// TIA Portal project "SCL_V13_SP1_1" (V13)

(* hardware
DEVICE "ET 200S-Station_1"  ET 200S station
   slot 0: "Baugruppenträger_0"  Rail
   slot 2: "PLC_1"  IM151-8 CPU  6ES7 151-8AB00-0AB0  V2.7
      slot 1: "PROFINET-Schnittstelle_1"  PN-IO
         slot 1: "Port_1"  Port
         slot 2: "Port_2"  Port
         slot 3: "Port_3"  Port
   slot 4: "PM-E DC24V_1"  PM-E 24VDC  6ES7 138-4CA01-0AA0
   slot 5: "4AI x I 2WIRE ST_1"  4AI x I 2WIRE ST  6ES7 134-4GD00-0AB0
   slot 6: "2AO x U ST_1"  2AO x U ST  6ES7 135-4FB01-0AB0
   slot 7: "8DI x DC24V_1"  8DI x 24VDC  6ES7 131-4BF00-0AA0
   slot 8: "8DI x DC24V_2"  8DI x 24VDC  6ES7 131-4BF00-0AA0
   slot 9: "8DI x DC24V_3"  8DI x 24VDC  6ES7 131-4BF00-0AA0
   slot 10: "8DI x DC24V_4"  8DI x 24VDC  6ES7 131-4BF00-0AA0
   slot 11: "8DO x DC24V / 0,5A_1"  8DO x 24VDC / 0.5A  6ES7 132-4BF00-0AA0
   slot 12: "8DO x DC24V / 0,5A_2"  8DO x 24VDC / 0.5A  6ES7 132-4BF00-0AA0
   slot 13: "8DO x DC24V / 0,5A_3"  8DO x 24VDC / 0.5A  6ES7 132-4BF00-0AA0
   slot 14: "8DO x DC24V / 0,5A_4"  8DO x 24VDC / 0.5A  6ES7 132-4BF00-0AA0
DEVICE "HMI_1"  TP 177B 6" PN/DP
   slot 0: "HMI"  HMI  6AV6 642-0BA01-1AX1  11.0.2.0
   slot 1: "HMI_RT_1"  TP 177B 6" PN/DP  6AV6 642-0BA01-1AX1  11.0.2.0
   slot 5: "HMI_1.IE_CP_1"  PROFINET Schnittstelle
      slot 1: "PROFINET Schnittstelle_1"  PROFINET Schnittstelle
         slot 1: "Port_1"  Port
   slot 7: "HMI_1.MPI/DP_CP_1"  MPI/DP Schnittstelle
DEVICE "PC-System_1"  SIMATIC PC station
   slot 0: "SIMATIC PC-Station"  Rail  SIMATIC PC-Station  V1.0
      slot 125: "Stationmanager"  Station_Manager  V6.0.4
   slot 1: "IE Allgemein_1"  IE General  IE_CP  V8.2.0
   slot 2: "HMI_RT_2"  WinCC RT Advanced  6AV2 104-0xxxx-xxxx  13.0.0.0
*)

// ===== PLC "PLC_1"  IM151-8 CPU =====

VAR_GLOBAL   // PLC tag table "Standard-Variablentabelle"
   "Volumen_Kugel" AT %MD10 : Real;
   "Tag_1" AT %MD20 : Real;
   "Sensor" AT %EW272 : Int;
   "Zu_gross" AT %M3.0 : Bool;
   "Abstand" AT %MD60 : Real;
   "Bit" AT %M0.0 : Bool;
   "Status_scale" AT %MW64 : Word;
   "Test" AT %MD66 : Real;
   "Zaehleingang" AT %E3.0 : Bool;
   "Ueber_PV" AT %M0.1 : Bool;
   "Zaehlerausgang" AT %MW26 : Int;
END_VAR

DATA_BLOCK "Datenbaustein_1"   // DB1
{ S7_Optimized_Access := 'FALSE' }
VERSION : 0.1
   VAR
      Datenspeicher : Array[1..2, 1..10] of Real;
   END_VAR
BEGIN
END_DATA_BLOCK

DATA_BLOCK "Daten_lesen_schreiben_DB"   // DB2
{ S7_Optimized_Access := 'FALSE' }
VERSION : 0.1
// stored: InstanceOfName Daten_lesen_schreiben
"Daten_lesen_schreiben"
BEGIN
END_DATA_BLOCK

FUNCTION_BLOCK "Daten_lesen_schreiben"   // FB1, SCL
{ S7_Optimized_Access := 'FALSE' }
VERSION : 0.1
BEGIN
   IF #Index <1 THEN
       #Index := 1; END_IF;
   IF #Index >10 THEN
       #Index := 10; END_IF;
   IF #Schreiben = true THEN
       #Daten[1, #Index] := #Druck;
       #Daten[2, #Index] := #Menge;
   ELSE
       #Druck := #Daten[1, #Index];
       #Menge := #Daten[2, #Index];
   END_IF;
END_FUNCTION_BLOCK

FUNCTION "Kugelvolumen" : Void   // FC1, SCL
{ S7_Optimized_Access := 'FALSE' }
VERSION : 0.1
BEGIN

   #Kugelvolumen := 3.14 *4 /3 * "Baustein_1"(Exponent := 3, Zahl := (#Durchmesser / 2));
   // Bei der unteren Formel gibt es ein falsches Ergebnis -> Immer probieren!
   //#Kugelvolumen := 4 / 3 * 3.14 * "Exponent"(Exponenten := 3, Zahl := (#Durchmesser / 2));
END_FUNCTION

FUNCTION "Exponent" : Void   // FC2, SCL
{ S7_Optimized_Access := 'FALSE' }
VERSION : 0.1
BEGIN
   IF #Exponenten >= 1 THEN
       #Ergebnis := 1;
       FOR #n := 1 TO #Exponenten DO
           // Statement section FOR
           #Ergebnis := #Zahl * #Ergebnis;
       END_FOR;
       #Exponent := #Ergebnis;
   ELSE
       #Exponent := -1;
   END_IF;
END_FUNCTION

FUNCTION "Baustein_1" : Void   // FC3, SCL
{ S7_Optimized_Access := 'FALSE' }
VERSION : 0.1
BEGIN
   IF #Exponent >= 1 THEN
       #Zwischenergebnis := 1;
       //Kommentar
       FOR #n := 1 TO #Exponent DO
           #Zwischenergebnis := #Zwischenergebnis * #Zahl;
       END_FOR;
       #Baustein_1 := #Zwischenergebnis;
   ELSE
       #Baustein_1 := -1;
   END_IF;
END_FUNCTION

FUNCTION "Abstand_rechnen" : Void   // FC4, SCL
{ S7_Optimized_Access := 'FALSE' }
VERSION : 0.1
BEGIN
   .0IF (#Sensor_Eingang > -4800) THEN
       // Statement section IF
       #Abstand_rechnen:=(#Sensor_Eingang-56)*-4.0/4856;
       #Zu_gross := false;
   ELSE
       #Abstand_rechnen := -1;
       #Zu_gross := true;
   END_IF;
END_FUNCTION

ORGANIZATION_BLOCK "Main"   // OB1, FBD
TITLE = "Main Program Sweep (Cycle)"
{ S7_Optimized_Access := 'FALSE' }
VERSION : 0.1
BEGIN

REGION Network 1
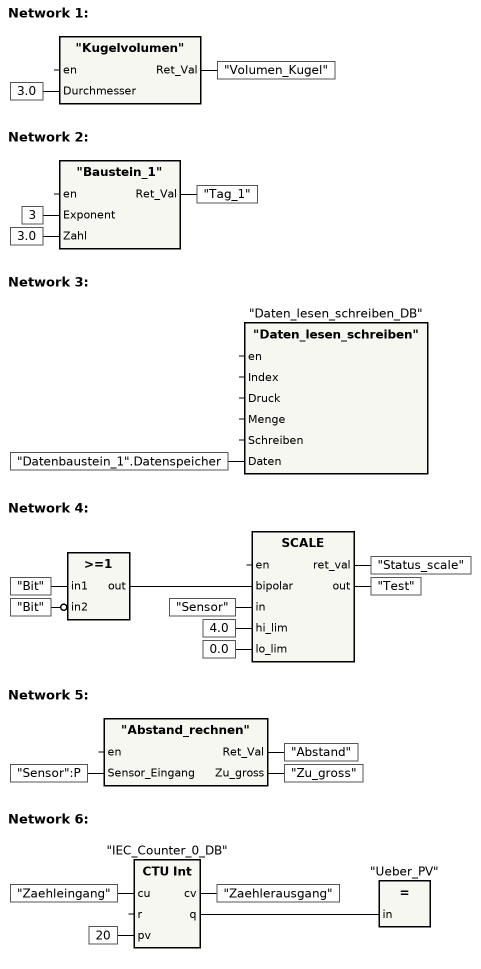
   "Volumen_Kugel" := "Kugelvolumen"(Durchmesser := 3.0);
END_REGION

REGION Network 2
   "Tag_1" := "Baustein_1"(Exponent := 3, Zahl := 3.0);
END_REGION

REGION Network 3
   "Daten_lesen_schreiben_DB"(Daten := "Datenbaustein_1".Datenspeicher);   // "Daten_lesen_schreiben"
END_REGION

REGION Network 4
   "Status_scale" := SCALE(bipolar := "Bit" OR NOT "Bit",
                           in := "Sensor",
                           hi_lim := 4.0,
                           lo_lim := 0.0,
                           out => "Test");
END_REGION

REGION Network 5
   "Abstand" := "Abstand_rechnen"(Sensor_Eingang := "Sensor":P, Zu_gross => "Zu_gross");
END_REGION

REGION Network 6
   "IEC_Counter_0_DB".CTU(cu := "Zaehleingang", pv := 20, cv => "Zaehlerausgang");
   "Ueber_PV" := "IEC_Counter_0_DB".q;
END_REGION
END_ORGANIZATION_BLOCK

(* ===== HMI "HMI_RT_1" =====
connection "HMI_Verbindung_1": ETHERNET, SIMATIC S7 300/400 MPI

HMI tags "Standard-Variablentabelle"
   "Daten_lesen_schreiben_DB_Druck" : Real, 1 s
   "Daten_lesen_schreiben_DB_Menge" : Real, 1 s
   "Daten_lesen_schreiben_DB_Schreiben" : Bool, 1 s
   "Daten_lesen_schreiben_DB_Index" : Int, 1 s
   "Abstand" : Real = PLC "Abstand", 1 s
   "Zu_gross" : Bool = PLC "Zu_gross", 1 s

screen "Bild_1" 320x240
   IOField "EA-Feld_1" at 168,39 size 107x20
   IOField "EA-Feld_2" at 168,78 size 108x20
   Button "Schaltfläche_1" at 195,116 size 80x25
   TextField "Textfeld_1" at 109,39 size 36x20
   TextField "Textfeld_2" at 109,78 size 42x20
   IOField "EA-Feld_3" at 191,164 size 80x20
   Button "Schaltfläche_2" at 190,193 size 44x25
   Button "Schaltfläche_3" at 234,193 size 44x25
   Button "Schaltfläche_4" at 0,213 size 160x25

screen "Bild_2" 320x240
   TextField "Textfeld_1" at 17,63 size 97x20
   Button "Schaltfläche_1" at 5,211 size 160x25
   Gauge "Zeigerinstrument_1" at 164,10 size 149x149
*)